SUBAPPLICATION Reset (* Subapplication Type *)
  (* Standard: 61499-2 *)
  (* Version 1.0, 2023-02-17, Franz *)
  IMPORT isobus::UT::Q::const::IDs::ID_NULL;
  IMPORT isobus::UT::io::Button::ButtonActivationCode::BT_RELEASED_UNLATCHED;
  IMPORT isobus::UT::io::Softkey::SoftKeyActivationCode::SK_RELEASED;
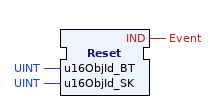
  EVENT_OUTPUT
    IND;
  END_EVENT
  VAR_INPUT
    u16ObjId_BT : UINT := ID_NULL; (* Object ID Button *)
    u16ObjId_SK : UINT := ID_NULL; (* Object ID SoftKey *)
  END_VAR
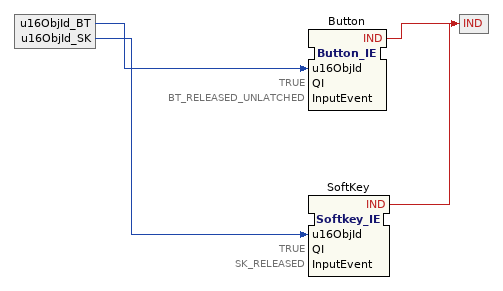
  FBS
    Button : isobus::UT::io::Button::Button_IE(QI := TRUE, InputEvent := BT_RELEASED_UNLATCHED);
    SoftKey : isobus::UT::io::Softkey::Softkey_IE(QI := TRUE, InputEvent := SK_RELEASED);
  END_FBS
  EVENT_CONNECTIONS
    Button.IND TO IND;
    SoftKey.IND TO IND;
  END_CONNECTIONS
  DATA_CONNECTIONS
    u16ObjId_BT TO Button.u16ObjId;
    u16ObjId_SK TO SoftKey.u16ObjId;
  END_CONNECTIONS
END_SUBAPPLICATION
